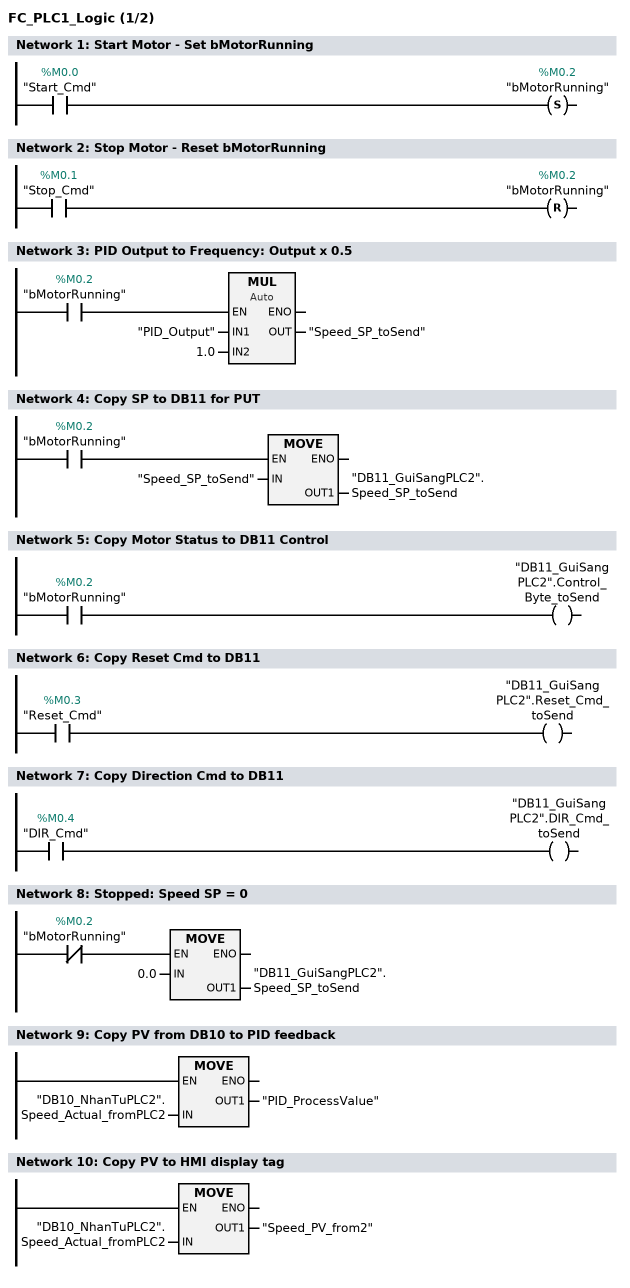
   RUNG wire#powerrail
      Contact( "Start_Cmd" )
      S_Coil( "bMotorRunning" )
   END_RUNG
   // the same network as SCL:
   IF "Start_Cmd" THEN "bMotorRunning" := TRUE; END_IF;
END_REGION

REGION Network 2: Stop Motor - Reset bMotorRunning
   RUNG wire#powerrail
      Contact( "Stop_Cmd" )
      R_Coil( "bMotorRunning" )
   END_RUNG
   // the same network as SCL:
   IF "Stop_Cmd" THEN "bMotorRunning" := FALSE; END_IF;
END_REGION

REGION Network 3: PID Output to Frequency: Output x 0.5
   RUNG wire#powerrail
      Contact( "bMotorRunning" )
      { S7_GenerateENO := "TRUE" } Mul(in1 := "PID_Output", in2 := 1.0, out => "Speed_SP_toSend")
   END_RUNG
   // the same network as SCL:
   IF "bMotorRunning" THEN "Speed_SP_toSend" := "PID_Output" * 1.0; END_IF;
END_REGION

REGION Network 4: Copy SP to DB11 for PUT
   RUNG wire#powerrail
      Contact( "bMotorRunning" )
      { S7_GenerateENO := "TRUE" } Move(in := "Speed_SP_toSend", out1 => "DB11_GuiSangPLC2".Speed_SP_toSend)
   END_RUNG
   // the same network as SCL:
   IF "bMotorRunning" THEN "DB11_GuiSangPLC2".Speed_SP_toSend := "Speed_SP_toSend"; END_IF;
END_REGION

REGION Network 5: Copy Motor Status to DB11 Control
   RUNG wire#powerrail
      Contact( "bMotorRunning" )
      Coil( "DB11_GuiSangPLC2".Control_Byte_toSend )
   END_RUNG
   // the same network as SCL:
   "DB11_GuiSangPLC2".Control_Byte_toSend := "bMotorRunning";
END_REGION

REGION Network 6: Copy Reset Cmd to DB11
   RUNG wire#powerrail
      Contact( "Reset_Cmd" )
      Coil( "DB11_GuiSangPLC2".Reset_Cmd_toSend )
   END_RUNG
   // the same network as SCL:
   "DB11_GuiSangPLC2".Reset_Cmd_toSend := "Reset_Cmd";
END_REGION

REGION Network 7: Copy Direction Cmd to DB11
   RUNG wire#powerrail
      Contact( "DIR_Cmd" )
      Coil( "DB11_GuiSangPLC2".DIR_Cmd_toSend )
   END_RUNG
   // the same network as SCL:
   "DB11_GuiSangPLC2".DIR_Cmd_toSend := "DIR_Cmd";
END_REGION

REGION Network 8: Stopped: Speed SP = 0
   RUNG wire#powerrail
      I_Contact( "bMotorRunning" )
      { S7_GenerateENO := "TRUE" } Move(in := 0.0, out1 => "DB11_GuiSangPLC2".Speed_SP_toSend)
   END_RUNG
   // the same network as SCL:
   IF NOT "bMotorRunning" THEN "DB11_GuiSangPLC2".Speed_SP_toSend := 0.0; END_IF;
END_REGION

REGION Network 9: Copy PV from DB10 to PID feedback
   RUNG wire#powerrail
      { S7_GenerateENO := "TRUE" } Move(in := "DB10_NhanTuPLC2".Speed_Actual_fromPLC2, out1 => "PID_ProcessValue")
   END_RUNG
   // the same network as SCL:
   "PID_ProcessValue" := "DB10_NhanTuPLC2".Speed_Actual_fromPLC2;
END_REGION

REGION Network 10: Copy PV to HMI display tag
   RUNG wire#powerrail
      { S7_GenerateENO := "TRUE" } Move(in := "DB10_NhanTuPLC2".Speed_Actual_fromPLC2, out1 => "Speed_PV_from2")
   END_RUNG
   // the same network as SCL:
   "Speed_PV_from2" := "DB10_NhanTuPLC2".Speed_Actual_fromPLC2;
END_REGION

REGION Network 11: Copy ATV12 Status to HMI tag
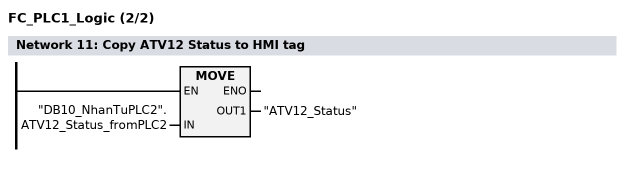
   RUNG wire#powerrail
      { S7_GenerateENO := "TRUE" } Move(in := "DB10_NhanTuPLC2".ATV12_Status_fromPLC2, out1 => "ATV12_Status")
   END_RUNG
   // the same network as SCL:
   "ATV12_Status" := "DB10_NhanTuPLC2".ATV12_Status_fromPLC2;
END_REGION
END_FUNCTION

FUNCTION "FC_PLC2_Logic" : Void   // FC10, LAD
{ S7_Optimized_Access := 'TRUE' }
VERSION : 0.1
// stored: AutoNumber true, IsIECCheckEnabled false, SetENOAutomatically false, UDAEnableTagReadback false
BEGIN

REGION Network 1: Freq Scale: SP x 10
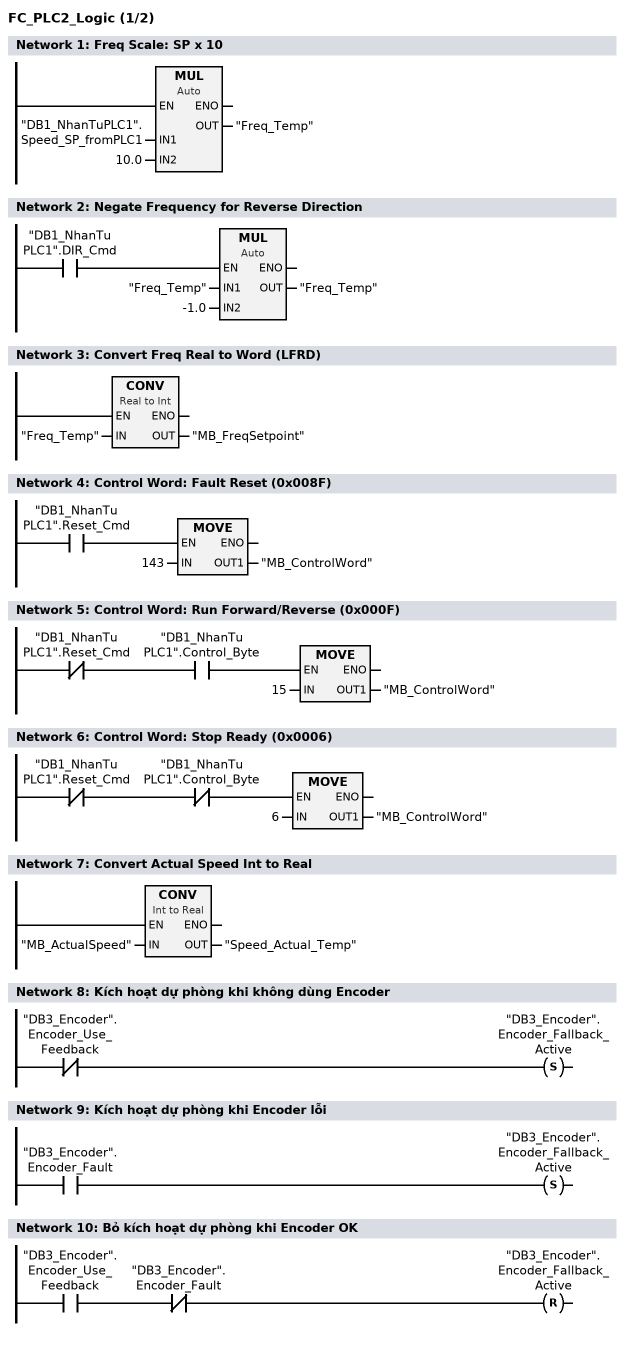
   RUNG wire#powerrail
      { S7_GenerateENO := "TRUE" } Mul(in1 := "DB1_NhanTuPLC1".Speed_SP_fromPLC1, in2 := 10.0, out => "Freq_Temp")
   END_RUNG
   // the same network as SCL:
   "Freq_Temp" := "DB1_NhanTuPLC1".Speed_SP_fromPLC1 * 10.0;
END_REGION

REGION Network 2: Negate Frequency for Reverse Direction
   RUNG wire#powerrail
      Contact( "DB1_NhanTuPLC1".DIR_Cmd )
      { S7_GenerateENO := "TRUE" } Mul(in1 := "Freq_Temp", in2 := -1.0, out => "Freq_Temp")
   END_RUNG
   // the same network as SCL:
   IF "DB1_NhanTuPLC1".DIR_Cmd THEN "Freq_Temp" := "Freq_Temp" * (-1.0); END_IF;
END_REGION

REGION Network 3: Convert Freq Real to Word (LFRD)
   RUNG wire#powerrail
      { S7_Templates := "[SrcType := Real, DestType := Int]"; S7_GenerateENO := "TRUE" } Convert(in := "Freq_Temp", out => "MB_FreqSetpoint")
   END_RUNG
   // the same network as SCL:
   "MB_FreqSetpoint" := REAL_TO_INT("Freq_Temp");
END_REGION

REGION Network 4: Control Word: Fault Reset (0x008F)
   RUNG wire#powerrail
      Contact( "DB1_NhanTuPLC1".Reset_Cmd )
      { S7_GenerateENO := "TRUE" } Move(in := 143, out1 => "MB_ControlWord")
   END_RUNG
   // the same network as SCL:
   IF "DB1_NhanTuPLC1".Reset_Cmd THEN "MB_ControlWord" := 143; END_IF;
END_REGION

REGION Network 5: Control Word: Run Forward/Reverse (0x000F)
   RUNG wire#powerrail
      I_Contact( "DB1_NhanTuPLC1".Reset_Cmd )
      Contact( "DB1_NhanTuPLC1".Control_Byte )
      { S7_GenerateENO := "TRUE" } Move(in := 15, out1 => "MB_ControlWord")
   END_RUNG
   // the same network as SCL:
   IF NOT "DB1_NhanTuPLC1".Reset_Cmd AND "DB1_NhanTuPLC1".Control_Byte THEN "MB_ControlWord" := 15; END_IF;
END_REGION

REGION Network 6: Control Word: Stop Ready (0x0006)
   RUNG wire#powerrail
      I_Contact( "DB1_NhanTuPLC1".Reset_Cmd )
      I_Contact( "DB1_NhanTuPLC1".Control_Byte )
      { S7_GenerateENO := "TRUE" } Move(in := 6, out1 => "MB_ControlWord")
   END_RUNG
   // the same network as SCL:
   IF NOT "DB1_NhanTuPLC1".Reset_Cmd AND NOT "DB1_NhanTuPLC1".Control_Byte THEN
       "MB_ControlWord" := 6;
   END_IF;
END_REGION

REGION Network 7: Convert Actual Speed Int to Real
   RUNG wire#powerrail
      { S7_Templates := "[SrcType := Int, DestType := Real]"; S7_GenerateENO := "TRUE" } Convert(in := "MB_ActualSpeed", out => "Speed_Actual_Temp")
   END_RUNG
   // the same network as SCL:
   "Speed_Actual_Temp" := INT_TO_REAL("MB_ActualSpeed");
END_REGION

REGION Network 8: Kích hoạt dự phòng khi không dùng Encoder
   RUNG wire#powerrail
      I_Contact( "DB3_Encoder".Encoder_Use_Feedback )
      S_Coil( "DB3_Encoder".Encoder_Fallback_Active )
   END_RUNG
   // the same network as SCL:
   IF NOT "DB3_Encoder".Encoder_Use_Feedback THEN "DB3_Encoder".Encoder_Fallback_Active := TRUE; END_IF;
END_REGION

REGION Network 9: Kích hoạt dự phòng khi Encoder lỗi
   RUNG wire#powerrail
      Contact( "DB3_Encoder".Encoder_Fault )
      S_Coil( "DB3_Encoder".Encoder_Fallback_Active )
   END_RUNG
   // the same network as SCL:
   IF "DB3_Encoder".Encoder_Fault THEN "DB3_Encoder".Encoder_Fallback_Active := TRUE; END_IF;
END_REGION

REGION Network 10: Bỏ kích hoạt dự phòng khi Encoder OK
   RUNG wire#powerrail
      Contact( "DB3_Encoder".Encoder_Use_Feedback )
      I_Contact( "DB3_Encoder".Encoder_Fault )
      R_Coil( "DB3_Encoder".Encoder_Fallback_Active )
   END_RUNG
   // the same network as SCL:
   IF "DB3_Encoder".Encoder_Use_Feedback AND NOT "DB3_Encoder".Encoder_Fault THEN
       "DB3_Encoder".Encoder_Fallback_Active := FALSE;
   END_IF;
END_REGION

REGION Network 11: Gửi tốc độ thực về PLC_1 chế độ bình thường
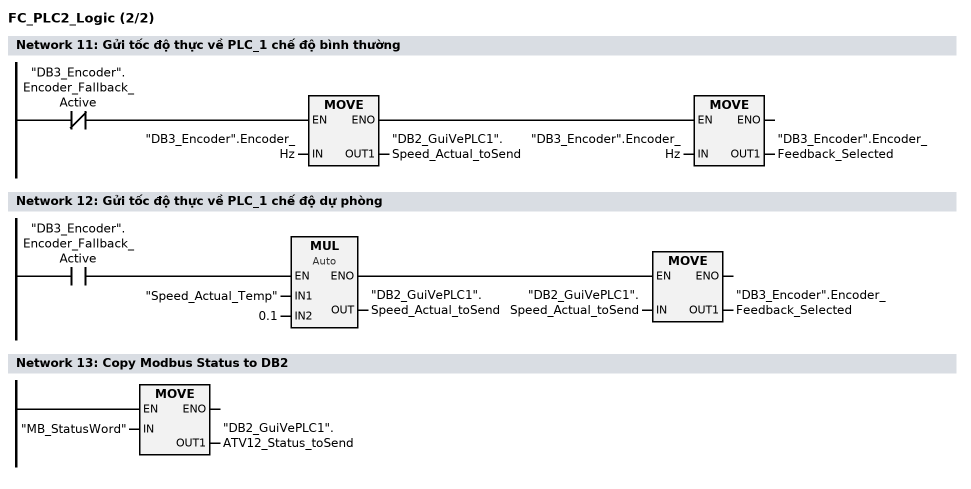
   RUNG wire#powerrail
      I_Contact( "DB3_Encoder".Encoder_Fallback_Active )
      { S7_GenerateENO := "TRUE" } Move(in := "DB3_Encoder".Encoder_Hz, out1 => "DB2_GuiVePLC1".Speed_Actual_toSend)
      { S7_GenerateENO := "TRUE" } Move(in := "DB3_Encoder".Encoder_Hz, out1 => "DB3_Encoder".Encoder_Feedback_Selected)
   END_RUNG
   // the same network as SCL:
   // ENO of a box is taken as its EN; it also drops when the box reports an error
   IF NOT "DB3_Encoder".Encoder_Fallback_Active THEN
       "DB2_GuiVePLC1".Speed_Actual_toSend := "DB3_Encoder".Encoder_Hz;
       "DB3_Encoder".Encoder_Feedback_Selected := "DB3_Encoder".Encoder_Hz;
   END_IF;
END_REGION

REGION Network 12: Gửi tốc độ thực về PLC_1 chế độ dự phòng
   RUNG wire#powerrail
      Contact( "DB3_Encoder".Encoder_Fallback_Active )
      { S7_GenerateENO := "TRUE" } Mul(in1 := "Speed_Actual_Temp", in2 := 0.1, out => "DB2_GuiVePLC1".Speed_Actual_toSend)
      { S7_GenerateENO := "TRUE" } Move(in := "DB2_GuiVePLC1".Speed_Actual_toSend, out1 => "DB3_Encoder".Encoder_Feedback_Selected)
   END_RUNG
   // the same network as SCL:
   // ENO of a box is taken as its EN; it also drops when the box reports an error
   IF "DB3_Encoder".Encoder_Fallback_Active THEN
       "DB2_GuiVePLC1".Speed_Actual_toSend := "Speed_Actual_Temp" * 0.1;
       "DB3_Encoder".Encoder_Feedback_Selected := "DB2_GuiVePLC1".Speed_Actual_toSend;
   END_IF;
END_REGION

REGION Network 13: Copy Modbus Status to DB2
   RUNG wire#powerrail
      { S7_GenerateENO := "TRUE" } Move(in := "MB_StatusWord", out1 => "DB2_GuiVePLC1".ATV12_Status_toSend)
   END_RUNG
   // the same network as SCL:
   "DB2_GuiVePLC1".ATV12_Status_toSend := "MB_StatusWord";
END_REGION
END_FUNCTION

FUNCTION "MHJ-PLC-Lab-Function-S71200" : Void   // FC9000, SCL
{ S7_Optimized_Access := 'TRUE' }
VERSION : 0.1
// stored: AutoNumber false, IsIECCheckEnabled false, SetENOAutomatically false, UDAEnableTagReadback false
   VAR_TEMP
      rdTimeReturn : Int;
      outputTime : DTL;
      SyncVal : Byte;
      forVal : Int;
      forVal_2 : Int;
      Value : Byte;
   END_VAR
   VAR CONSTANT
      CompVal : Byte := 16#34;
      Value_01 : Byte := 16#11;
      Value_01_DW : DWord := 16#A165_D992;
      Value_02_DW : DWord := 16#58BE_4401;
   END_VAR
BEGIN

   #Value:=PEEK(area := 16#82,
        dbNumber := 0,
        byteOffset := 511);
   #Value := #Value + 1;

   POKE(area := 16#82,
        dbNumber := 0,
        byteOffset := 511,
        value := #Value);

   POKE(area:=16#81,
        dbNumber:=0,
        byteOffset:=1016,
        value:=#Value_01_DW);
   POKE(area := 16#81,
        dbNumber := 0,
        byteOffset := 1020,
        value := #Value_02_DW);

   POKE(area := 16#81,
        dbNumber := 0,
        byteOffset := 511,
        value := B#16#00);

   FOR #forVal := 0 TO 120 DO
       FOR #forVal_2:=0 TO 10 DO
           #rdTimeReturn:=RD_SYS_T(#outputTime);
           #rdTimeReturn := WR_SYS_T(#outputTime);
           #rdTimeReturn := RD_SYS_T(#outputTime);
           #rdTimeReturn := WR_SYS_T(#outputTime);
       END_FOR;
       #SyncVal:= PEEK(area := 16#81,
                      dbNumber := 0,
                      byteOffset := 511);
       IF #SyncVal = #CompVal THEN
          GOTO M_1;
       END_IF;
   END_FOR;
   RETURN;

   M_1:
   POKE(area := 16#81,
        dbNumber := 0,
        byteOffset := 511,
        value := B#16#0);
END_FUNCTION

FUNCTION_BLOCK "PID"   // FB1, SCL
{ S7_Optimized_Access := 'TRUE' }
VERSION : 0.1
// stored: AutoNumber true, IsIECCheckEnabled false, IsRetainMemResEnabled false, MemoryReserve 100, SetENOAutomatically false, UDAEnableTagReadback false
   VAR_INPUT
      ki : Real := 0.002;
      kp : Real := 11.0;
      kd : Real;
      level : Real;
      setpoint : Real;
      drain : Bool;
      "full drain" : Bool;
      emergency : Bool;
   END_VAR
   VAR_OUTPUT
      filling : Real;
      draining : Real;
      errordisplay : Real;
      setpointdisplay : DInt;
      leveldisplay : DInt;
   END_VAR
   VAR
      integralop : Real;
      oldintegral : Real;
      err2 : Real;
   END_VAR
   VAR_TEMP
      error : Real;
      u : Real;
      temp : DInt;
   END_VAR
BEGIN

   #errordisplay := ABS(#setpoint - #level);

   //display setpoint to 100%
   #setpointdisplay := REAL_TO_DINT(#setpoint*10.0);
   //



   //display level to 100%
   #leveldisplay :=REAL_TO_DINT( #level*10.0);
   //
   #temp := REAL_TO_DINT(#kp);

   #error := #setpoint - #level;

   #integralop := #integralop + #error; //sums all the past errors to present error
   #u := (#error * #kp) + (#integralop * (#ki / 10)) + (#kd * (#err2 - #error));
   #filling := #u;
   #draining := -#u;


   //if error always goes up the filling will always goes up
   //and it will be more that 100% .but the valve can go only to 100% open
   //so if it goes up.we stop the valve at 10 and  stabilized the integral
   IF (#filling > 10.0) THEN
       #integralop := #oldintegral;
       #filling := 10.0;
   END_IF;
   //same thing but for values under 0
   IF (#filling < 0.0) THEN
       #integralop := #oldintegral;
       #filling := 0.0;
   END_IF;
   IF (#draining > 10.0) THEN
       #integralop := #oldintegral;
       #draining := 10.0;
   END_IF;

   IF (#draining < 0.0) THEN
       #integralop := #oldintegral;
       #draining := 0.0;
   END_IF;

   #oldintegral := #integralop; //past error sum
   #err2 := #error;//past error

   IF #drain THEN
       #draining := 10.0;

   END_IF;

   IF #"full drain" THEN
       #draining := 10.0;
       #filling := 0;
   END_IF;
   IF #emergency THEN
       #draining := 0;
       #filling := 0;

   END_IF;
END_FUNCTION_BLOCK

DATA_BLOCK "Timer_Sim_DB"   // DB10
TITLE = Timer_Sim_DB
// Instance DB for simulation timer
// stored: AutoNumber true, InstanceOfName IEC_TIMER, OfSystemLibElement IEC_TIMER, OfSystemLibVersion 1.0
"IEC_TIMER"
   // VAR
   //    PT : Time;
   //    ET { ExternalWritable := 'False'} : Time;
   //    IN : Bool;
   //    Q { ExternalWritable := 'False'} : Bool;
   // END_VAR
BEGIN
END_DATA_BLOCK

DATA_BLOCK "MB_SERVER_DB"   // DB53
// stored: AutoNumber true, DBAccessibleFromOPCUA true, InstanceOfName MB_SERVER_3, OfSystemLibElement MB_SERVER, OfSystemLibVersion 3.1
"MB_SERVER_3"
   // VAR_INPUT
   //    DISCONNECT : Bool;
   //    CONNECT_ID : UInt;
   //    IP_PORT : UInt;
   // END_VAR
   // VAR_OUTPUT
   //    NDR : Bool;
   //    DR : Bool;
   //    ERROR : Bool;
   //    STATUS : Word;
   // END_VAR
   // VAR_IN_OUT
   //    MB_HOLD_REG : Variant;
   // END_VAR
   // VAR
   //    TCON_SFB { S7_SetPoint := 'True'} : TCON;
   //    TDISCON_SFB { S7_SetPoint := 'True'} : TDISCON;
   //    TSEND_SFB { S7_SetPoint := 'True'} : TSEND;
   //    TRCV_SFB { S7_SetPoint := 'True'} : TRCV;
   //    TCON_Param { S7_SetPoint := 'True'} : TCON_Param;
   //    MB_State : UInt;
   //    Request_Count : UInt;
   //    Server_Message_Count : UInt;
   //    Xmt_Rcv_Count : UInt;
   //    Exception_Count : UInt;
   //    Success_Count : UInt;
   //    SL_Status_Hold : UInt;
   //    HR_Start_Offset : UInt;
   //    Init_OK : Bool;
   //    SL_Error_State : Bool;
   //    Connected : Bool;
   //    XMT_Set_NDR : Bool;
   //    XMT_Set_DR : Bool;
   // END_VAR
BEGIN
END_DATA_BLOCK

DATA_BLOCK "MB_CLIENT_DB"   // DB52
// stored: AutoNumber false, DBAccessibleFromOPCUA true, InstanceOfName MB_CLIENT, OfSystemLibElement MB_CLIENT, OfSystemLibVersion 3.1
"MB_CLIENT"
   // VAR_INPUT
   //    REQ : Bool;
   //    DISCONNECT : Bool;
   //    CONNECT_ID : UInt;
   //    IP_OCTET_1 : USInt;
   //    IP_OCTET_2 : USInt;
   //    IP_OCTET_3 : USInt;
   //    IP_OCTET_4 : USInt;
   //    IP_PORT : UInt;
   //    MB_MODE : USInt;
   //    MB_DATA_ADDR : UDInt;
   //    MB_DATA_LEN : UInt;
   // END_VAR
   // VAR_OUTPUT
   //    DONE : Bool;
   //    BUSY : Bool;
   //    ERROR : Bool;
   //    STATUS : Word;
   // END_VAR
   // VAR_IN_OUT
   //    MB_DATA_PTR : Variant;
   // END_VAR
   // VAR
   //    TCON_SFB { S7_SetPoint := 'True'} : TCON;
   //    TDISCON_SFB { S7_SetPoint := 'True'} : TDISCON;
   //    TSEND_SFB { S7_SetPoint := 'True'} : TSEND;
   //    TRCV_SFB { S7_SetPoint := 'True'} : TRCV;
   //    TCON_PARAM { S7_SetPoint := 'True'} : TCON_Param;
   //    PF_FREQUENCY : Real;
   //    BLOCKED_PROC_TIMEOUT : Real;
   //    RCV_TIMEOUT : Real;
   //    CURRENT_TIME_VALUE : DWord;
   //    SAVED_TIME_VALUE : DWord;
   //    XMT_TIME : DWord;
   //    SAVED_CONNECT_ID : Word;
   //    SAVED_IP_PORT : Word;
   //    SAVED_MODE : Byte;
   //    SAVED_IP1 : Byte;
   //    SAVED_IP2 : Byte;
   //    SAVED_IP3 : Byte;
   //    SAVED_IP4 : Byte;
   //    SAVED_DATA_ADDR : DWord;
   //    SAVED_DATA_LEN : Word;
   //    MB_STATE : Word;
   //    COMM_SENT_COUNT : Word;
   //    BYTE_COUNT : Word;
   //    BYTE_COUNTB : Byte;
   //    SAVED_START_ADDR : Word;
   //    MB_TRANSACTION_ID : Word;
   //    MB_UNIT_ID : Word;
   //    RETRIES : Word;
   //    INIT_OK : Bool;
   //    ACTIVE : Bool;
   //    CONNECTED : Bool;
   //    SAVED_MA_REQ : Bool;
   // END_VAR
BEGIN
   TCON_PARAM.CONNECTION_TYPE := 11;
   TCON_PARAM.LOCAL_DEVICE_ID := 64;
END_DATA_BLOCK

DATA_BLOCK "MB_COMM_LOAD_DB"   // DB50
// stored: AutoNumber false, DBAccessibleFromOPCUA true, InstanceOfName MB_COMM_LOAD, OfSystemLibElement MB_COMM_LOAD, OfSystemLibVersion 2.1
"MB_COMM_LOAD"
   // VAR_INPUT
   //    REQ : Bool;
   //    PORT : PORT;
   //    BAUD : UDInt;
   //    PARITY : UInt;
   //    FLOW_CTRL : UInt;
   //    RTS_ON_DLY : UInt;
   //    RTS_OFF_DLY : UInt;
   //    RESP_TO : UInt;
   // END_VAR
   // VAR_OUTPUT
   //    DONE : Bool;
   //    ERROR : Bool;
   //    STATUS : Word;
   // END_VAR
   // VAR_IN_OUT
   //    MB_DB : MB_BASE;
   // END_VAR
   // VAR
   //    ICHAR_GAP : UInt;
   //    RETRIES : UInt;
   //    WRREC_STATUS : Word;
   //    RDREC_STATUS : Word;
   //    SFC_STATUS : Word;
   //    Port_CFG_SFB : Array[0..25] of Byte;
   //    Send_CFG_SFB : Array[0..16] of Byte;
   //    Rcv_CFG_SFB : Array[0..60] of Byte;
   //    STOP_BITS : USInt;
   // END_VAR
BEGIN
END_DATA_BLOCK

DATA_BLOCK "MB_MASTER_DB"   // DB51
// stored: AutoNumber false, DBAccessibleFromOPCUA true, InstanceOfName MB_MASTER, OfSystemLibElement MB_MASTER, OfSystemLibVersion 2.2
"MB_MASTER"
   // // inherited from MB_BASE
   // VAR
   //    S_PORT : UInt;
   //    S_RESP_TO : UInt;
   //    S_ICHAR_GAP : UInt;
   //    S_RETRIES : UInt;
   // END_VAR
   // VAR_INPUT
   //    REQ : Bool;
   //    MB_ADDR : UInt;
   //    MODE : USInt;
   //    DATA_ADDR : UDInt;
   //    DATA_LEN : UInt;
   // END_VAR
   // VAR_OUTPUT
   //    DONE : Bool;
   //    BUSY : Bool;
   //    ERROR : Bool;
   //    STATUS : Word;
   // END_VAR
   // VAR_IN_OUT
   //    DATA_PTR : Variant;
   // END_VAR
   // VAR
   //    SEND_PTP_SFB : Array[0..11] of Byte;
   //    RCV_PTP_SFB : Array[0..11] of Byte;
   //    RCV_RST_SFB : Array[0..9] of Byte;
   //    PF_FREQUENCY : Real;
   //    BLOCKED_PROC_TIMEOUT : Real;
   //    CURRENT_TIME_VALUE : UDInt;
   //    SAVED_TIME_VALUE : UDInt;
   //    SAVED_SLAVE_ADDR : Word;
   //    SAVED_MODE : Word;
   //    SAVED_DATA_ADDR : DWord;
   //    SAVED_DATA_LEN : UInt;
   //    MB_STATE : UInt;
   //    COMM_SENT_COUNT : UInt;
   //    BYTE_COUNT : USInt;
   //    INIT_OK : Bool;
   //    ACTIVE : Bool;
   //    BROADCAST_FLAG : Bool;
   //    EXTENDED_ADDRESSING : Bool;
   //    SAVED_START_ADDR : UInt;
   //    TXBuf_Function_Offset : UDInt;
   //    TXBuf_Address_Offset : UDInt;
   //    TXBuf_Quantity_Offset : UDInt;
   // END_VAR
BEGIN
END_DATA_BLOCK

DATA_BLOCK "PID_DB"   // DB6
VERSION : 0.1
// stored: AutoNumber true, InstanceOfName PID, InstanceOfType FB
"PID"
BEGIN
END_DATA_BLOCK

DATA_BLOCK "PI_DB"   // DB3
VERSION : 0.1
// stored: AutoNumber true, InstanceOfName PID, InstanceOfType FB
"PID"
BEGIN
END_DATA_BLOCK
